{attribute 'GeneratedUsingTerminal: EK1100-0000-0018'}
{attribute addProperty BoxType "EK1100-0000-0018"}
{attribute addProperty Id "Term_234_EL1809EL1809_32157CFD20"}
{attribute addProperty CRC "3412413499"}
{attribute addProperty Size "20"}
{attribute addProperty Name "Term 233 (EK1100)"}
TYPE Term_233_EK1100_CB654C3B EXTENDS EK1100_1FC0878B :
STRUCT
	{attribute addProperty Name "Term 234 (EL1809)"}
	{attribute addProperty PreviousPort "Term 233 (EK1100) : B"}
	{attribute addProperty SyncUnit "default"}
	Term_234_EL1809 : EL1809_32157CFD;
END_STRUCT
END_TYPE

(* stored: Version 1.2.0.0, ProductVersion 3.1.4024.11
   DUT Term_233_EK1100_CB654C3B: Id {e934e9a0-6224-481e-b1c5-6e7df6ae51a9} *)
